// TwinCAT 3 PLC project AssertionTests
// ProgramVersion: 3.1.4026.19
// libraries:
//   CNM_AbstractObject, * (ekvip automation GmbH)
//   CNM_AssertionInterfaces, * (ekvip automation GmbH)
//   CNM_AssertionInterfaceTests, * (ekvip automation GmbH)
//   CNM_ReturnTypes, * (ekvip automation GmbH)
//   Tc2_Standard, * (Beckhoff Automation GmbH)
//   Tc2_System, * (Beckhoff Automation GmbH)
//   Tc3_Module, * (Beckhoff Automation GmbH)
//   TcUnit, * (www.tcunit.org)
// project tree:
//   ConcreteAssertions/ ConcreteAssertions.TcPOU
//   MainTask/ MAIN.TcPOU, PlcTask.TcTTO (not stored)
// real-time tasks:
//   TASK PlcTask: cycle T#10ms, priority 20, ADS port 350
//   TASK CNC-Task ADS: cycle default, priority 7, ADS port 558
//   TASK CNC-Task COM: cycle T#10ms, priority 13, ADS port 556
//   TASK CNC-Task SDA: cycle T#10ms, priority 8, ADS port 555
//   TASK CNC-Task GEO: cycle T#2ms, priority 3, ADS port 554

// ---- ConcreteAssertions/ConcreteAssertions.TcPOU
FUNCTION_BLOCK ConcreteAssertions EXTENDS CNM_AssertionInterfaces.AbstractAssertor IMPLEMENTS CNM_AssertionInterfaceTests.IAssertorContainer
VAR
	wrongAssertion	:BOOL;
END_VAR

METHOD assertionWasWrong
VAR_INPUT
	caller			:CNM_AbstractObject.IObject;
	message			:CNM_AssertionInterfaces.AssertMessage;
	additionalText	:Tc2_System.T_MaxString;
END_VAR
THIS^.wrongAssertion := TRUE;
END_METHOD

PROPERTY assertor : CNM_AssertionInterfaces.IAssertor
GET
assertor := THIS^;
END_GET
END_PROPERTY

PROPERTY className : CNM_AbstractObject.ClassName
GET
className := 'ConcreteAssertions';
END_GET
END_PROPERTY

METHOD resetAssertor
THIS^.wasAssertionWrong := FALSE;
END_METHOD

PROPERTY wasAssertionWrong : BOOL
GET
wasAssertionWrong := THIS^.wrongAssertion;
END_GET
SET
THIS^.wrongAssertion := wasAssertionWrong;
END_SET
END_PROPERTY

END_FUNCTION_BLOCK

// ---- MainTask/MAIN.TcPOU
PROGRAM MAIN
VAR
	concrete				:ConcreteAssertions();
	tests					:CNM_AssertionInterfaceTests.AssertionTester(concrete);
END_VAR

TcUnit.RUN_IN_SEQUENCE();

END_PROGRAM
